TYPE ST_ModuleStatus :
STRUCT
	ModuleId : UDINT;
	Enabled : BOOL;
	IsControlSourceAlive : BOOL;
	Configuration : ST_ModuleConfigurationStatus;
	ResponseId : UDINT;
	PackMLOut : ST_PML_Base_Out;
	Alarm : ST_ModuleAlarmStatus;
	Data : ST_ModuleDataStatus;
END_STRUCT
END_TYPE

(* stored: Version 1.1.0.1, ProductVersion 3.1.4026.18
   DUT ST_ModuleStatus: Id {6c7acf88-b8e8-4b23-b4ca-30b3cf9d6905} *)
